PROGRAM PRG_LoadcellScaling
VAR
	bActivateLoadcellScaling AT %I*: BOOL;
	bDeactivateLoadcellScaling AT %I*:BOOL;
	bActiveState: BOOL;
	bZeroing: BOOL;
	bSet300Gr: BOOL;
	nMinValue: DINT:=430;
	nMaxValue: DINT:=1100;
END_VAR

// Detect /deactivate state for function 
IF 	bActivateLoadcellScaling AND NOT bDeactivateLoadcellScaling THEN
	bActiveState:=TRUE;
ELSIF 	bDeactivateLoadcellScaling AND NOT bActivateLoadcellScaling THEN
	bActiveState:=FALSE;
END_IF

// Funtion execute
IF bActiveState THEN
	IF bZeroing THEN
		nMinValue:= GVL.uLoadCellRawValue;
	END_IF
	IF bSet300Gr THEN
		nMaxValue:= GVL.uLoadCellRawValue;
	END_IF
	GVL.uLoadCellScaledValue := F_Scale(GVL.uLoadCellRawValue, 0.0, 0.3, nMinValue, nMaxValue);
ELSE
	GVL.uLoadCellScaledValue:= 0.0;
END_IF

END_PROGRAM

(* stored: Version 1.1.0.1, ProductVersion 3.1.4024.12
   POU PRG_LoadcellScaling: Id {976f5398-c837-4944-8db6-b5f1f3ab8dcc}, SpecialFunc None *)
